TYPE "Positioning_MOL_Machine_CIn"
VERSION : 0.1
// Block: Positioning_MOL_Machine_CIn
   STRUCT
      Manager : Positioning_MOL_Machine_Manager;
      MinusExtEnable : Bool;
      PlusExtEnable : Bool;
      ExternalAlarms : Bool;
      PositionLimits : Struct
         EnableMin : Bool;
         PosMin : LReal;
         EnableMax : Bool;
         PosMax : LReal;
      END_STRUCT;
   END_STRUCT;

END_TYPE
